DATA_BLOCK "ST10_Flow1_A1TableScan_iDB"
{ S7_Optimized_Access := 'TRUE' }
VERSION : 0.1
NON_RETAIN
"ST10_Flow1_A1TableScan"

BEGIN

END_DATA_BLOCK

